FUNCTION FGetMinimum : TIME
VAR_INPUT
	Times : ARRAY[1..10] OF TIME;
END_VAR
VAR
	i : INT;
	MinVal : TIME;
END_VAR

MinVal := Times[1];

FOR i := 2 TO 10 DO
	IF Times[i] < MinVal THEN
		MinVal := Times[i];
	END_IF
END_FOR;

FGetMinimum := MinVal;

END_FUNCTION

(* stored: Version 1.1.0.1, ProductVersion 3.1.4024.15
   POU FGetMinimum: Id {1a92f618-e780-43d5-8559-73ac5ae17d57}, SpecialFunc None *)
